# EPICS substitutions: iocBoot/iocoh26/substitutions/motor.substitutions
file "$(MOTOR)/motorApp/Db/asyn_motor.db"
{
pattern
{N,        M,         DTYP,        PORT,  ADDR,           DESC,    EGU,  DIR,  VELO,  VBAS,  ACCL,  BDST,  BVEL,  BACC,   MRES,  PREC,  DHLM,  DLLM,  INIT,  RTRY}
{1,  "m$(N)",  "asynMotor",  "ANG1_1_1",     0,  "AMCI ANG1 1",  "deg",  Pos,     1,     0,    .2,     0,    50,    .2,  0.002,     2,   1e9,  -1e9,    "",     0}
}
